FUNCTION_BLOCK FB_Object EXTENDS TcLog
VAR_INPUT
	bBool					: BOOL;
END_VAR
VAR
	Logger					: FB_EventLogger();
	
END_VAR

IF bBool THEN
	Logger.Append('Io ')
	.Append('sono ')
	.Debug('Batman');
ELSE
	Logger.CanSpam()
	.Append('Io ')
	.Append('sono ')
	.Debug('Superman');
END_IF

END_FUNCTION_BLOCK

(* stored: Version 1.1.0.1, ProductVersion 3.1.4024.12
   POU FB_Object: Id {069a147d-2605-4c5a-b1b5-85f9f72aa0b5}, SpecialFunc None *)
